// Mitsubishi GX Works2 project: 0625(SM4xx이용한 점멸)   PLC: Q02/Q02H

PROGRAM MAIN
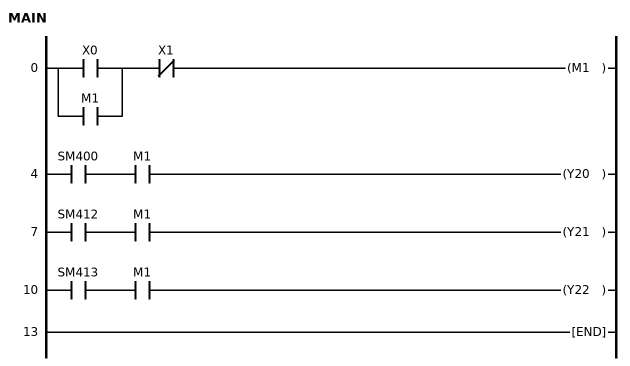
0     LD      X0
      OR      M1
      ANI     X1
      OUT     M1
4     LD      SM400
      AND     M1
      OUT     Y20
7     LD      SM412
      AND     M1
      OUT     Y21
10    LD      SM413
      AND     M1
      OUT     Y22
13    END
END_PROGRAM
